Universal Robots PolyScope program: program3.urp

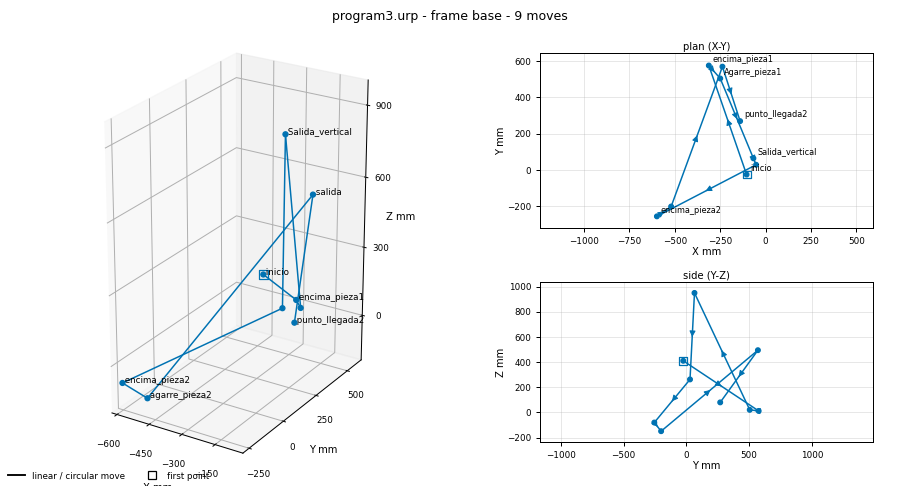
[picture p0: tool path of program3.urp in frame base, 9 of 9 moves have a stored position in this frame; points joined in program order, loops and branches not executed]
Program program3 (installation=default directory=/ursim/programs createdIn=3.15.8.106339 lastSavedIn=3.15.8.106339 robotSerialNumber=2018359999)
Calibrated DH parameters: a=[0, -0.425, -0.39225, 0, 0, 0]; d=[0.089159, 0, 0, 0.10915, 0.09465, 0.0823]; alpha=[1.570796, 0, 0, 1.570796, -1.570796, 0]; deltaTheta=[0, 0, 0, 0, 0, 0]
Robot Program (runOnlyOnce=false)
  MoveJ speed 60 deg/s, acceleration 80 deg/s^2 (useActiveTCP=true)
    Waypoint inicio: TCP in base x=-104.438 y=-24.654 z=411.336 mm, rx=-0.395 ry=2.7386 rz=-1.1343 rad; joints [-72.577, -6.481, -131.082, -87.083, 91.477, 1.626] deg
    Loop Forever
      MoveL speed 250 mm/s, acceleration 1200 mm/s^2 (useActiveTCP=true) feature=Base
        Waypoint encima_pieza1: TCP in base x=-312.415 y=575.705 z=12.299 mm, rx=-0.6797 ry=-2.113 rz=-1.8952 rad; joints [-67.443, -43.609, 86.093, -32.995, 120.263, 32.428] deg
      MoveL speed 250 mm/s, acceleration 1200 mm/s^2 (useActiveTCP=true) feature=Base
        Waypoint Agarre_pieza1: TCP in base x=-249.52 y=504.424 z=21.145 mm, rx=1.2742 ry=1.9925 rz=1.6425 rad; joints [-67.443, -43.609, 86.093, 0.375, 151.341, 58.739] deg
      Set DigitalOutput (payload=1 tcpAsCog=true) pin=digital_out[0]; digitalValue=1
      MoveL speed 250 mm/s, acceleration 1200 mm/s^2 (useActiveTCP=true) feature=Base
        Waypoint Salida_vertical: TCP in base x=-66.885 y=64.744 z=951.339 mm, rx=-1.0936 ry=0.4819 rz=-1.4756 rad; joints [-67.443, -83.946, -13.19, 0.375, 151.341, 58.739] deg
      MoveL speed 250 mm/s, acceleration 1200 mm/s^2 (useActiveTCP=true) feature=Base
        Waypoint Waypoint_4: TCP in base x=-52.065 y=29.162 z=263.03 mm, rx=-1.742 ry=-0.6079 rz=-1.7823 rad; joints [-57.376, -151.968, 143.023, -7.261, 169.888, 77.9] deg
      Set DigitalOutput (payload=0 tcpAsCog=true) pin=digital_out[0]; digitalValue=0
      MoveL speed 250 mm/s, acceleration 1200 mm/s^2 (useActiveTCP=true) feature=Base
        Waypoint encima_pieza2: TCP in base x=-598.333 y=-254.889 z=-80.01 mm, rx=0.5643 ry=-2.0193 rz=-0.7167 rad; joints [17.146, -32.458, 77.97, -15.233, 120.673, 58.025] deg
      MoveL speed 250 mm/s, acceleration 1200 mm/s^2 (useActiveTCP=true) feature=Base
        Waypoint agarre_pieza2: TCP in base x=-519.939 y=-200.813 z=-148.97 mm, rx=-0.0107 ry=-2.2614 rz=-1.1585 rad; joints [17.146, -23.107, 77.97, 5.032, 149.001, 90.386] deg
        Set DigitalOutput pin=digital_out[0]; digitalValue=1
      MoveL speed 250 mm/s, acceleration 1200 mm/s^2 (useActiveTCP=true) feature=Base
        Waypoint salida: TCP in base x=-237.465 y=569.504 z=495.688 mm, rx=-1.4329 ry=-0.1875 rz=-1.5331 rad; joints [-70.952, -70.778, 62.019, -25.404, 149.001, 90.386] deg
      MoveL speed 250 mm/s, acceleration 1200 mm/s^2 (useActiveTCP=true) feature=Base
        Waypoint punto_llegada2: TCP in base x=-140.068 y=269.533 z=80.317 mm, rx=-1.192 ry=-1.6239 rz=-1.3505 rad; joints [-80.212, -88.655, 144.341, -43.281, 101.88, 72.784] deg
    Wait DigitalInput pin=digital_in[0]; digitalValue=0
